(* Logix 5000 project; controller ECHO_TEST5_V34 vendor 1 type 14 code 164 rev 35.11; software revision 35.00 *)

TASK MainTask (continuous, watchdog 500 ms) : MainProgram
TASK task300msp1 (periodic, rate 20 ms, priority 10, watchdog 500 ms) : MachineCtrl

MODULES
   Local : vendor 1 type 14 code 164 (ICP 0, rev 35.11)
END_MODULES

VAR_GLOBAL   (* controller tags *)
   ActualSpeed : DINT;
   ActualTemperature : REAL := 95.4;
   BatchName : STRING := 'Batch_117';
   FillingDelay : DINT := 1500;
   FillingPosition : REAL := 20.5;
   FillingPositionActaul : REAL;
   FillingTime : DINT := 1200;
   Humidity : DINT := 31;
   MachineRun : BOOL;
   MachineStart : BOOL;
   Pressure : REAL := 5.699477;
   SetSpeed : DINT := 100;
   SetTemperature : REAL := 100.0;
   Speed : DINT := 110;
   Temperature : REAL := 77.30285;
   TemperatureDeviation : REAL := 4.5999985;
   Triggertag : BOOL;
   Var1 : INT := 20;
   Var2 : DINT := 110;
   Var3 : REAL := 125.36;
   Var4 : STRING := 'Logic Comm Success';
   VarByte : USINT;
   VialType : STRING := '20 ml';
END_VAR

PROGRAM MachineCtrl   (* main routine MainRoutine *)
VAR
   FillingCompleted : BOOL;
   FillingDone : BOOL;
   FillingReady : BOOL;
   Timer1 : TIMER := (PRE := 1500);
   Timer2 : TIMER := (PRE := 1500);
END_VAR

ROUTINE MainRoutine   (* ladder *)
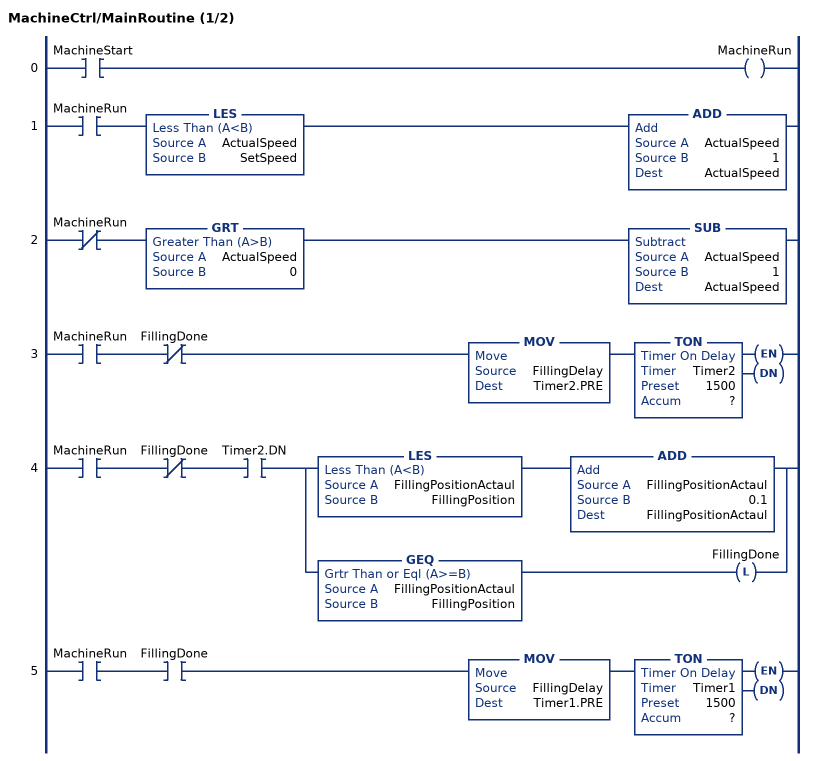
   0: XIC(MachineStart)OTE(MachineRun);
   1: XIC(MachineRun)LES(ActualSpeed,SetSpeed)ADD(ActualSpeed,1,ActualSpeed);
   2: XIO(MachineRun)GRT(ActualSpeed,0)SUB(ActualSpeed,1,ActualSpeed);
   3: XIC(MachineRun)XIO(FillingDone)MOV(FillingDelay,Timer2.PRE)TON(Timer2,?,?);
   4: XIC(MachineRun)XIO(FillingDone)XIC(Timer2.DN)[LES(FillingPositionActaul,FillingPosition) ADD(FillingPositionActaul,0.1,FillingPositionActaul) ,GEQ(FillingPositionActaul,FillingPosition) OTL(FillingDone) ];
   5: XIC(MachineRun)XIC(FillingDone)MOV(FillingDelay,Timer1.PRE)TON(Timer1,?,?);
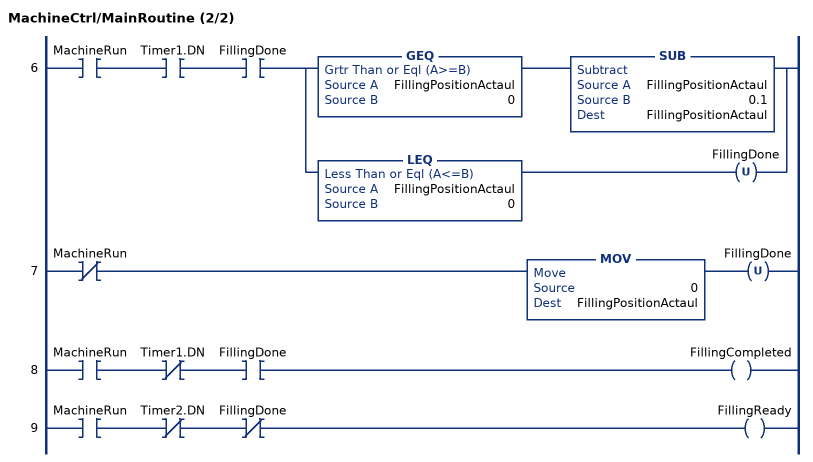
   6: XIC(MachineRun)XIC(Timer1.DN)XIC(FillingDone)[GEQ(FillingPositionActaul,0) SUB(FillingPositionActaul,0.1,FillingPositionActaul) ,LEQ(FillingPositionActaul,0) OTU(FillingDone) ];
   7: XIO(MachineRun)MOV(0,FillingPositionActaul)OTU(FillingDone);
   8: XIC(MachineRun)XIO(Timer1.DN)XIC(FillingDone)OTE(FillingCompleted);
   9: XIC(MachineRun)XIO(Timer2.DN)XIO(FillingDone)OTE(FillingReady);
END_ROUTINE
END_PROGRAM

PROGRAM MainProgram   (* main routine MainRoutine *)
VAR
   BatchNumber : DINT := 117;
   BatchNumberString : STRING := '117';
   BatchTestString : STRING := 'Batch_';
   HumidityIncDone : BOOL;
   LogVar1Counter : COUNTER := (PRE := 100, ACC := 84);
   LogVar2Counter : COUNTER := (PRE := 80, ACC := 44);
   LogVar3Counter : COUNTER := (PRE := 60, ACC := 13);
   LogVar4Counter : COUNTER := (PRE := 40, ACC := 33);
   ONSBITS : DINT := 256;
   PressureIncDone : BOOL;
   Run : BOOL;
   SpeedIncDone : BOOL := 1;
   Start : BOOL;
   TempDecDone : BOOL := 1;
   TempIncDone : BOOL;
   TempTimer : TIMER := (PRE := 4000, ACC := 3130, EN := 1, TT := 1);
   Timer1 : TIMER := (PRE := 3000, ACC := 1130, EN := 1, TT := 1);
   Timer2 : TIMER := (PRE := 1500, ACC := 1130, EN := 1, TT := 1);
END_VAR

ROUTINE MainRoutine   (* ladder *)
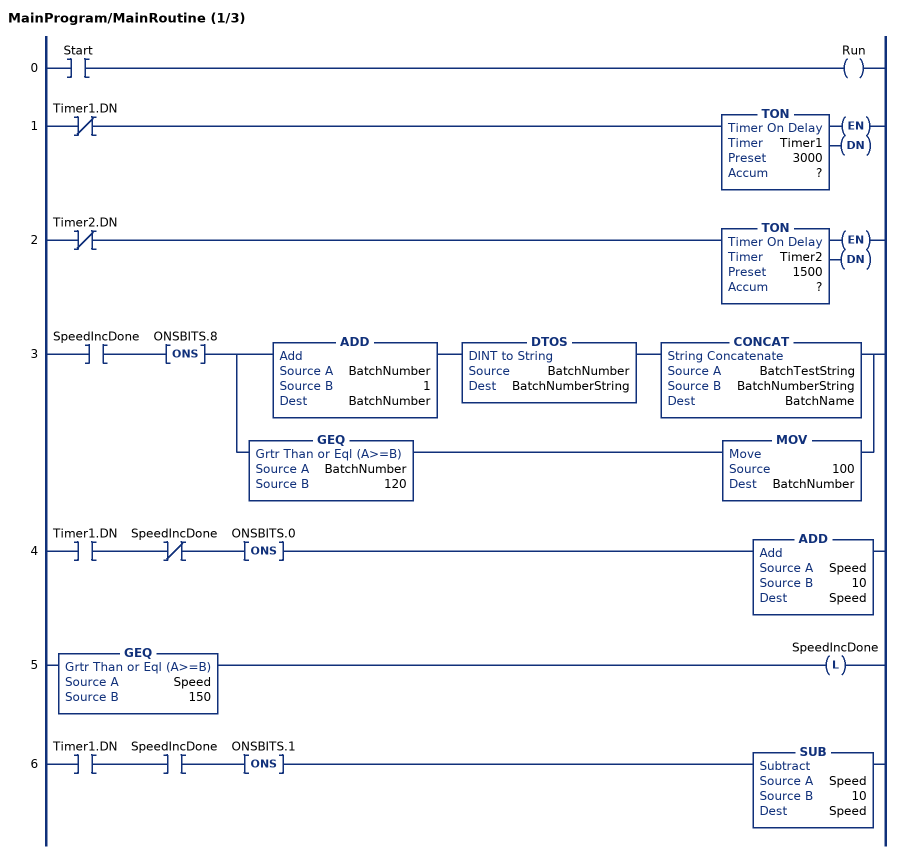
   0: XIC(Start)OTE(Run);
   1: XIO(Timer1.DN)TON(Timer1,?,?);
   2: XIO(Timer2.DN)TON(Timer2,?,?);
   3: XIC(SpeedIncDone)ONS(ONSBITS.8)[ADD(BatchNumber,1,BatchNumber) DTOS(BatchNumber,BatchNumberString) CONCAT(BatchTestString,BatchNumberString,BatchName) ,GEQ(BatchNumber,120) MOV(100,BatchNumber) ];
   4: XIC(Timer1.DN)XIO(SpeedIncDone)ONS(ONSBITS.0)ADD(Speed,10,Speed);
   5: GEQ(Speed,150)OTL(SpeedIncDone);
   6: XIC(Timer1.DN)XIC(SpeedIncDone)ONS(ONSBITS.1)SUB(Speed,10,Speed);
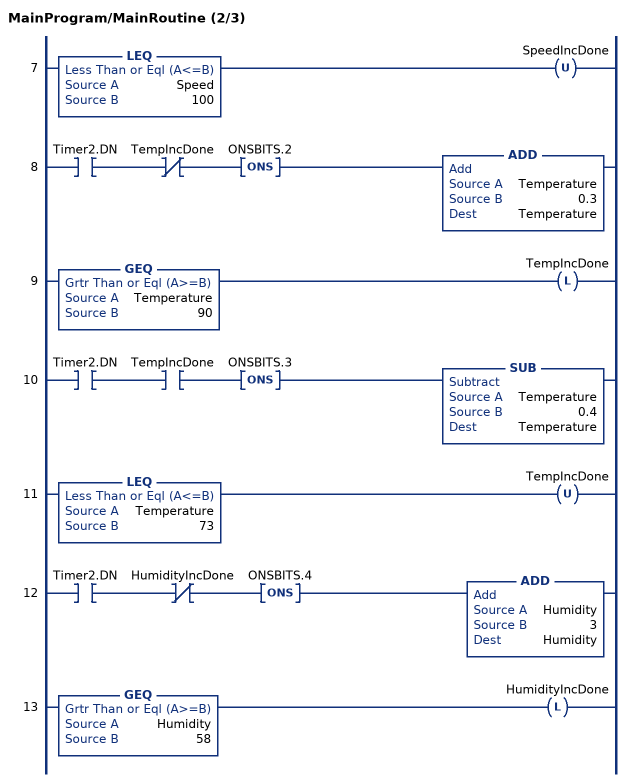
   7: LEQ(Speed,100)OTU(SpeedIncDone);
   8: XIC(Timer2.DN)XIO(TempIncDone)ONS(ONSBITS.2)ADD(Temperature,0.3,Temperature);
   9: GEQ(Temperature,90)OTL(TempIncDone);
   10: XIC(Timer2.DN)XIC(TempIncDone)ONS(ONSBITS.3)SUB(Temperature,0.4,Temperature);
   11: LEQ(Temperature,73)OTU(TempIncDone);
   12: XIC(Timer2.DN)XIO(HumidityIncDone)ONS(ONSBITS.4)ADD(Humidity,3,Humidity);
   13: GEQ(Humidity,58)OTL(HumidityIncDone);
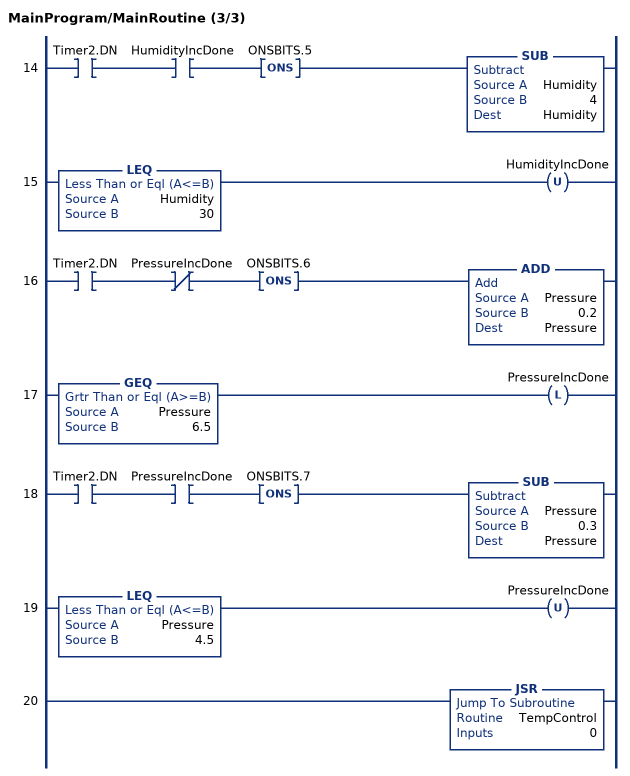
   14: XIC(Timer2.DN)XIC(HumidityIncDone)ONS(ONSBITS.5)SUB(Humidity,4,Humidity);
   15: LEQ(Humidity,30)OTU(HumidityIncDone);
   16: XIC(Timer2.DN)XIO(PressureIncDone)ONS(ONSBITS.6)ADD(Pressure,0.2,Pressure);
   17: GEQ(Pressure,6.5)OTL(PressureIncDone);
   18: XIC(Timer2.DN)XIC(PressureIncDone)ONS(ONSBITS.7)SUB(Pressure,0.3,Pressure);
   19: LEQ(Pressure,4.5)OTU(PressureIncDone);
   20: JSR(TempControl,0);
END_ROUTINE

ROUTINE TempControl   (* ladder *)
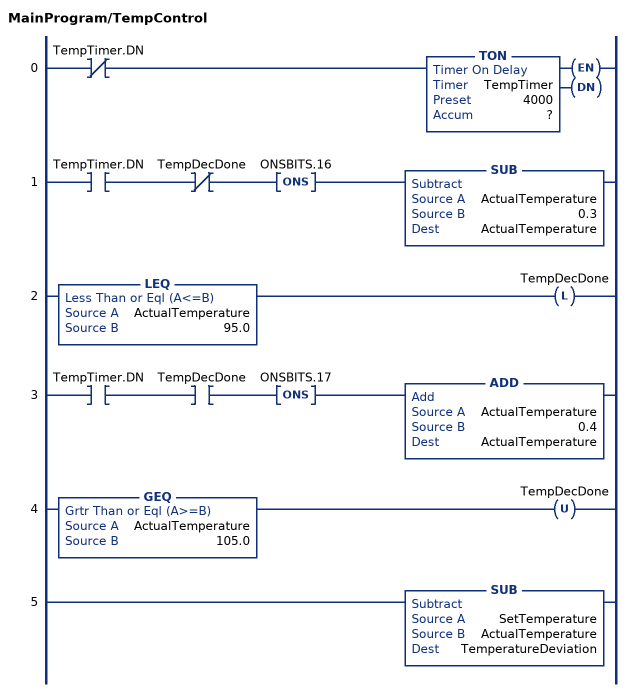
   0: XIO(TempTimer.DN)TON(TempTimer,?,?);
   1: XIC(TempTimer.DN)XIO(TempDecDone)ONS(ONSBITS.16)SUB(ActualTemperature,0.3,ActualTemperature);
   2: LEQ(ActualTemperature,95.0)OTL(TempDecDone);
   3: XIC(TempTimer.DN)XIC(TempDecDone)ONS(ONSBITS.17)ADD(ActualTemperature,0.4,ActualTemperature);
   4: GEQ(ActualTemperature,105.0)OTU(TempDecDone);
   5: SUB(SetTemperature,ActualTemperature,TemperatureDeviation);
END_ROUTINE
END_PROGRAM
